TYPE Cnv_Level_Control_DUT :
STRUCT
	Cnv1:	Buffer_Cnv_Control_DUT;
	Cnv2:	Buffer_Cnv_Control_DUT;
END_STRUCT
END_TYPE

(* stored: Version 1.1.0.1
   DUT Cnv_Level_Control_DUT: Id {4cb63c30-af5b-4d1d-ae3c-abbc2a710d54} *)
